FUNCTION WRITE_PROTECTED_REAL
VAR_INPUT
    Ptr : POINTER TO REAL;
    Value : REAL;
END_VAR

Ptr^ := Value;

END_FUNCTION

(* stored: Version 1.1.0.1, ProductVersion 3.1.4022.18
   POU WRITE_PROTECTED_REAL: Id {b51bba4d-2ead-4155-a62f-7a7ea20f8571}, SpecialFunc None *)
